// LS Electric XG5000 project: fda
// PLC LSPLC
// module base 0 slot 0: 입출력 모듈:XBC-DR32H (DC 24V 입력, 릴레이 출력 32점)
// module base 0 slot 1: 위치결정 모듈:XBF-PD02A (위치결정 펄스(LD)출력형, 2축)
// module base 0 slot 2: 출력 모듈:XBE-TN/TP16A (트랜지스터 출력, 16점 (싱크출력/소스출력))

PROGRAM NewProgram (task: 스캔 프로그램)

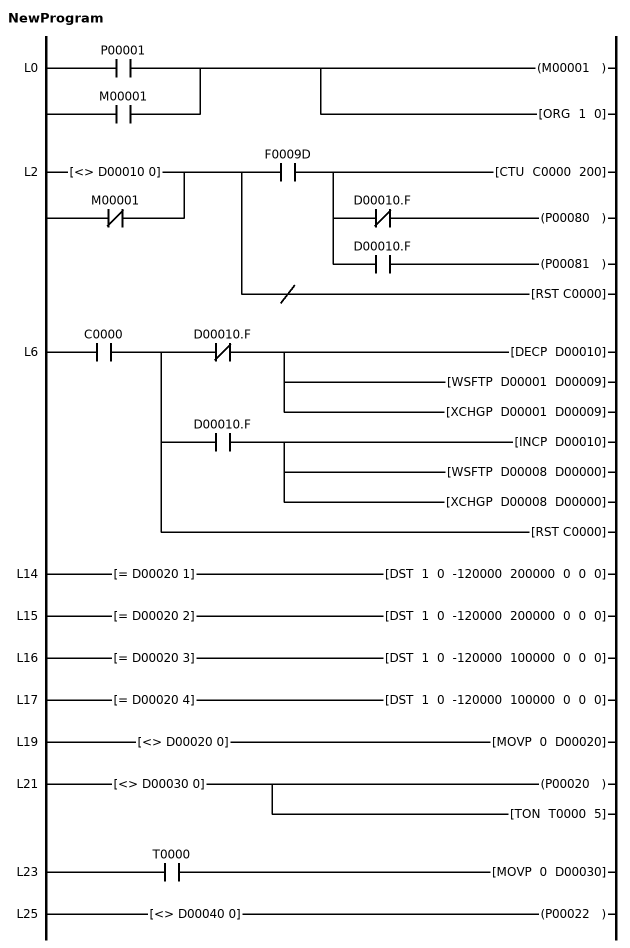
; L0
LOAD      P00001
OR        M00001
OUT       M00001
ORG       1 0
; L2
LOAD<>    D00010 0
OR NOT    M00001
MPUSH
AND       F0009D
CTU       C0000 200
MPUSH
AND NOT   D00010.F
OUT       P00080
MPOP
AND       D00010.F
OUT       P00081
MPOP
NOT
RST       C0000
; L6
LOAD      C0000
MPUSH
AND NOT   D00010.F
DECP      D00010
WSFTP     D00001 D00009
XCHGP     D00001 D00009
MLOAD
AND       D00010.F
INCP      D00010
WSFTP     D00008 D00000
XCHGP     D00008 D00000
MPOP
RST       C0000
; L14
LOAD=     D00020 1
DST       1 0 -120000 200000 0 0 0
; L15
LOAD=     D00020 2
DST       1 0 -120000 200000 0 0 0
; L16
LOAD=     D00020 3
DST       1 0 -120000 100000 0 0 0
; L17
LOAD=     D00020 4
DST       1 0 -120000 100000 0 0 0
; L19
LOAD<>    D00020 0
MOVP      0 D00020
; L21
LOAD<>    D00030 0
OUT       P00020
TON       T0000 5
; L23
LOAD      T0000
MOVP      0 D00030
; L25
LOAD<>    D00040 0
OUT       P00022